// TIA Portal V19 export
FUNCTION "A02_ButtonSafe_CALL" : Void   // FC184, LAD
TITLE = BUTTONS SAFE OF AREA 02 CALL
// stored: SetENOAutomatically false
BEGIN

REGION Network 1: LB114 Feed material of area 02
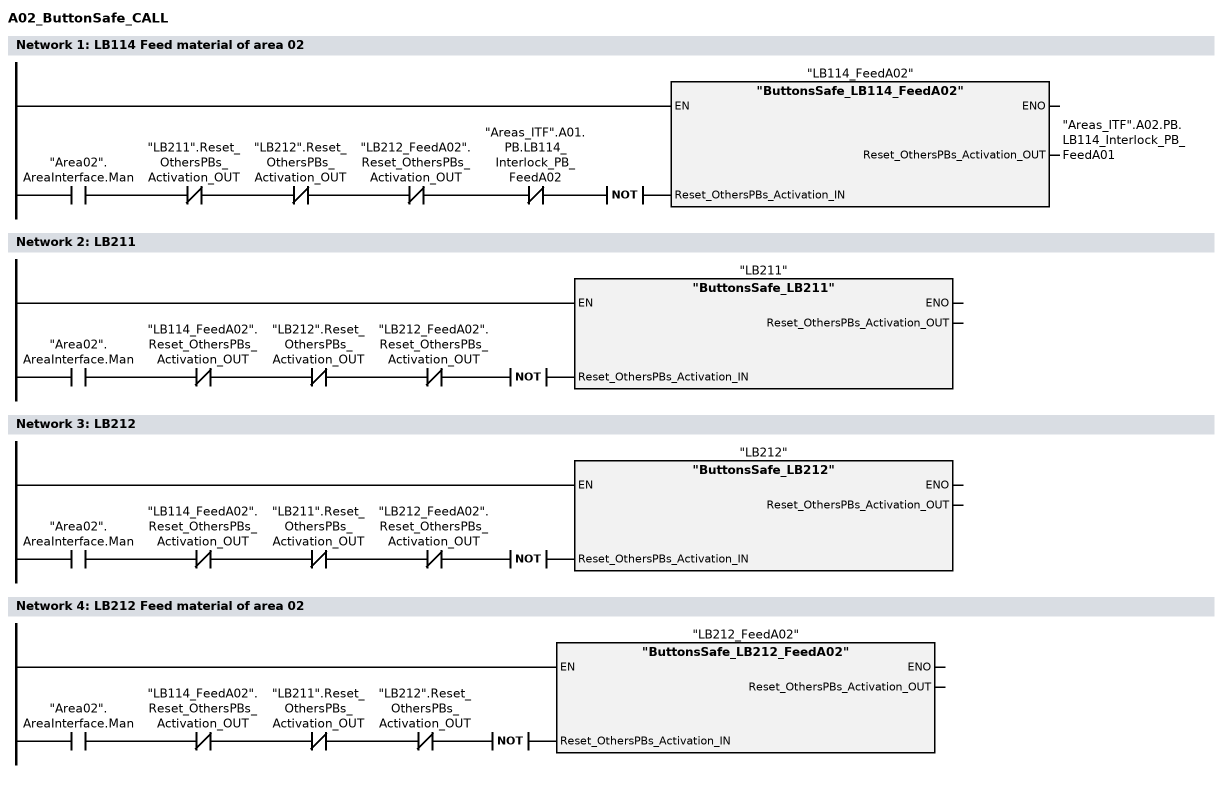
   RUNG wire#powerrail
      "LB114_FeedA02"(Reset_OthersPBs_Activation_IN := wire#w1, Reset_OthersPBs_Activation_OUT => "Areas_ITF".A02.PB.LB114_Interlock_PB_FeedA01)
   END_RUNG
   RUNG wire#powerrail
      Contact( "Area02".AreaInterface.Man )
      I_Contact( "LB211".Reset_OthersPBs_Activation_OUT )
      I_Contact( "LB212".Reset_OthersPBs_Activation_OUT )
      I_Contact( "LB212_FeedA02".Reset_OthersPBs_Activation_OUT )
      I_Contact( "Areas_ITF".A01.PB.LB114_Interlock_PB_FeedA02 )
      Not()
   END_RUNG wire#w1
   // the same network as SCL:
   "LB114_FeedA02"(Reset_OthersPBs_Activation_IN := NOT ("Area02".AreaInterface.Man AND NOT "LB211".Reset_OthersPBs_Activation_OUT AND NOT "LB212".Reset_OthersPBs_Activation_OUT AND NOT "LB212_FeedA02".Reset_OthersPBs_Activation_OUT AND NOT "Areas_ITF".A01.PB.LB114_Interlock_PB_FeedA02),   // "ButtonsSafe_LB114_FeedA02"
                   Reset_OthersPBs_Activation_OUT => "Areas_ITF".A02.PB.LB114_Interlock_PB_FeedA01);
END_REGION

REGION Network 2: LB211
   RUNG wire#powerrail
      "LB211"(Reset_OthersPBs_Activation_IN := wire#w1, Reset_OthersPBs_Activation_OUT =>)
   END_RUNG
   RUNG wire#powerrail
      Contact( "Area02".AreaInterface.Man )
      I_Contact( "LB114_FeedA02".Reset_OthersPBs_Activation_OUT )
      I_Contact( "LB212".Reset_OthersPBs_Activation_OUT )
      I_Contact( "LB212_FeedA02".Reset_OthersPBs_Activation_OUT )
      Not()
   END_RUNG wire#w1
   // the same network as SCL:
   "LB211"(Reset_OthersPBs_Activation_IN := NOT ("Area02".AreaInterface.Man AND NOT "LB114_FeedA02".Reset_OthersPBs_Activation_OUT AND NOT "LB212".Reset_OthersPBs_Activation_OUT AND NOT "LB212_FeedA02".Reset_OthersPBs_Activation_OUT));   // "ButtonsSafe_LB211"
END_REGION

REGION Network 3: LB212
   RUNG wire#powerrail
      "LB212"(Reset_OthersPBs_Activation_IN := wire#w1, Reset_OthersPBs_Activation_OUT =>)
   END_RUNG
   RUNG wire#powerrail
      Contact( "Area02".AreaInterface.Man )
      I_Contact( "LB114_FeedA02".Reset_OthersPBs_Activation_OUT )
      I_Contact( "LB211".Reset_OthersPBs_Activation_OUT )
      I_Contact( "LB212_FeedA02".Reset_OthersPBs_Activation_OUT )
      Not()
   END_RUNG wire#w1
   // the same network as SCL:
   "LB212"(Reset_OthersPBs_Activation_IN := NOT ("Area02".AreaInterface.Man AND NOT "LB114_FeedA02".Reset_OthersPBs_Activation_OUT AND NOT "LB211".Reset_OthersPBs_Activation_OUT AND NOT "LB212_FeedA02".Reset_OthersPBs_Activation_OUT));   // "ButtonsSafe_LB212"
END_REGION

REGION Network 4: LB212 Feed material of area 02
   RUNG wire#powerrail
      "LB212_FeedA02"(Reset_OthersPBs_Activation_IN := wire#w1, Reset_OthersPBs_Activation_OUT =>)
   END_RUNG
   RUNG wire#powerrail
      Contact( "Area02".AreaInterface.Man )
      I_Contact( "LB114_FeedA02".Reset_OthersPBs_Activation_OUT )
      I_Contact( "LB211".Reset_OthersPBs_Activation_OUT )
      I_Contact( "LB212".Reset_OthersPBs_Activation_OUT )
      Not()
   END_RUNG wire#w1
   // the same network as SCL:
   "LB212_FeedA02"(Reset_OthersPBs_Activation_IN := NOT ("Area02".AreaInterface.Man AND NOT "LB114_FeedA02".Reset_OthersPBs_Activation_OUT AND NOT "LB211".Reset_OthersPBs_Activation_OUT AND NOT "LB212".Reset_OthersPBs_Activation_OUT));   // "ButtonsSafe_LB212_FeedA02"
END_REGION
END_FUNCTION
